//==================================================================================================
//						Beckhoff Automation Poland
//							P_TaskInfo
//							15.11.2016
//
//				Program  odczytujący informacje o tasku
//
// 	v1.0 || TC v 3.1.4020.14 || - pierwsza wersja
//==================================================================================================
PROGRAM P_TaskInfo
VAR_OUTPUT
	bOK								: BOOL;	// Brak bledow i ostrzezen
	bWarning						: BOOL;	// Ostrzezenie - nie wystepuja w tym podprogramie - wystepuja dla zachowania spojnosci
	bError							: BOOL;	// Zbiorcza flaga bledow
	bReset							: BOOL; 
END_VAR
VAR
	fbTaskInfo						: FB_TaskInfo;
END_VAR

fbTaskInfo(bReset:=bReset , bError=> );
bError := fbTaskInfo.bError; // Dla jednego tasku. W przypadku wiekszej ilosci taskow trzeba dopisac reszte.

bOk := NOT bError;

END_PROGRAM

(* stored: Version 1.1.0.1, ProductVersion 3.1.4022.7
   POU P_TaskInfo: Id {963be1aa-f497-42e7-bc03-3e87922b27c9}, SpecialFunc None *)
